// TIA Portal V20 export
// export: Created 2025-12-01T14:56:58.9383901Z, ExportSetting None, DisplayName Totally Integrated Automation Portal, DisplayVersion V20 Update 3, DisplayName TIA Portal Openness, DisplayVersion V20 Update 3, DisplayName TIA Portal Version Control Interface, DisplayVersion V20 Update 3, DisplayName STEP 7 Professional, DisplayVersion V20 Update 3, DisplayName STEP 7 Safety, DisplayVersion V20 Update 2, DisplayName WinCC Basic/Comfort/Advanced, DisplayVersion V20 Update 3, DisplayName WinCC Professional, DisplayVersion V20 Update 3, DisplayName WinCC Unified, DisplayVersion V20 Update 3
FUNCTION_BLOCK "FB89_GALIBO_Remontada_EnRodillos"   // FB89, LAD
TITLE = Galibo de 5 Alturas (2023)
{ S7_Optimized_Access := 'FALSE' }
AUTHOR : GALIBO
NAME : 20140101
VERSION : 3.0
// stored: AutoNumber false, SetENOAutomatically false
   VAR_INPUT
      Mesa : UInt;
      NumGalibo : UInt;
      pHs_Remontado_1Dcha : Bool;
      pHs_Remontado_2Dcha : Bool;
      pHs_Remontado_1Izq : Bool;
      pHs_Remontado_2Izq : Bool;
      HabilitarLectura : Bool;
      PermisoLectura : Bool;
      Rearmar_ConMesaLibre : Bool;
      V_Estabilidad : Int;
   END_VAR
   VAR_OUTPUT
      Codigo : Word;
      FinLectura : Bool;
   END_VAR
   VAR_IN_OUT
      SinopticoGalibo_Señal : "UDT_HMI_SeñalesGalibo";
      SinopticoGalibo_Codigo : Word;
   END_VAR
   VAR
      CNT_Estabilidad : "FB910_CNT_UHS";
      GAL_ET00 : Bool;
      GAL_ET01 : Bool;
      GAL_ET02 : Bool;
      GAL_ET03 : Bool;
      pHsGalibo_OK { ExternalAccessible := 'False'; ExternalVisible := 'False'; ExternalWritable := 'False'} : Bool;
      LeerRemontado : Bool;
      FinRemontado : Bool;
      Remontado_NO : Bool;
      Remontado_SI : Bool;
      CodigoRemontado : SInt;
      MemoCodigo : Word;
      STAT_Baliza_Galibo : Bool;
   END_VAR
   VAR_TEMP
      EstadoZona : "EstadoZona";
      EstadoVI : "EstadosMesa";
   END_VAR
BEGIN

REGION Network 1: INICIALIZAR - Recoger las Variables de Estado de la Mesa
   // Se recoge - Estado_CBx
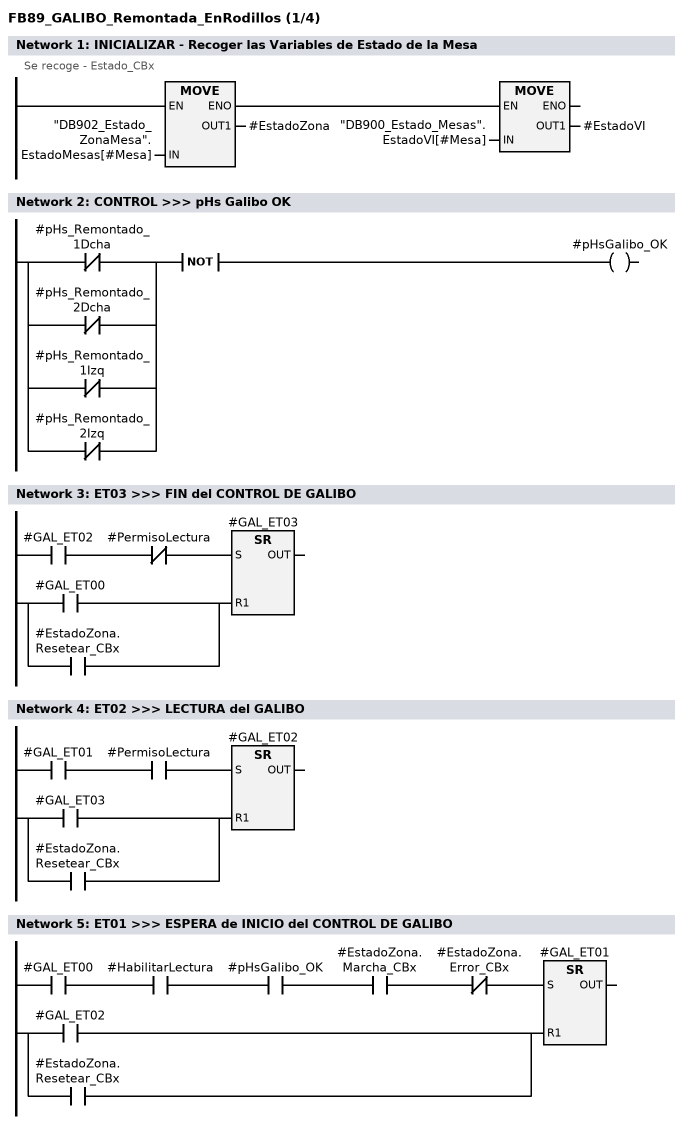
   RUNG wire#powerrail
      Move(in := "DB902_Estado_ZonaMesa".EstadoMesas[#Mesa], out1 => #EstadoZona)
      Move(in := "DB900_Estado_Mesas".EstadoVI[#Mesa], out1 => #EstadoVI)
   END_RUNG
   // the same network as SCL:
   #EstadoZona := "DB902_Estado_ZonaMesa".EstadoMesas[#Mesa];
   #EstadoVI := "DB900_Estado_Mesas".EstadoVI[#Mesa];
END_REGION

REGION Network 2: CONTROL >>> pHs Galibo OK
   RUNG wire#powerrail
      I_Contact( #pHs_Remontado_1Dcha )
      wire#w1
      Not()
      Coil( #pHsGalibo_OK )
   END_RUNG
   RUNG wire#powerrail
      I_Contact( #pHs_Remontado_2Dcha )
   END_RUNG wire#w1
   RUNG wire#powerrail
      I_Contact( #pHs_Remontado_1Izq )
   END_RUNG wire#w1
   RUNG wire#powerrail
      I_Contact( #pHs_Remontado_2Izq )
   END_RUNG wire#w1
   // the same network as SCL:
   #pHsGalibo_OK := NOT (NOT #pHs_Remontado_1Dcha OR NOT #pHs_Remontado_2Dcha OR NOT #pHs_Remontado_1Izq OR NOT #pHs_Remontado_2Izq);
END_REGION

REGION Network 3: ET03 >>> FIN del CONTROL DE GALIBO
   RUNG wire#powerrail
      Contact( #GAL_ET02 )
      I_Contact( #PermisoLectura )
      S_SR(operand := #GAL_ET03, r1 := wire#w1)
   END_RUNG
   RUNG wire#powerrail
      Contact( #GAL_ET00 )
   END_RUNG wire#w1
   RUNG wire#powerrail
      Contact( #EstadoZona.Resetear_CBx )
   END_RUNG wire#w1
   // the same network as SCL:
   IF #GAL_ET02 AND NOT #PermisoLectura THEN
       #GAL_ET03 := TRUE;   // SR flip-flop
   END_IF;
   IF #GAL_ET00 OR #EstadoZona.Resetear_CBx THEN #GAL_ET03 := FALSE; END_IF;
END_REGION

REGION Network 4: ET02 >>> LECTURA del GALIBO
   RUNG wire#powerrail
      Contact( #GAL_ET01 )
      Contact( #PermisoLectura )
      S_SR(operand := #GAL_ET02, r1 := wire#w1)
   END_RUNG
   RUNG wire#powerrail
      Contact( #GAL_ET03 )
   END_RUNG wire#w1
   RUNG wire#powerrail
      Contact( #EstadoZona.Resetear_CBx )
   END_RUNG wire#w1
   // the same network as SCL:
   IF #GAL_ET01 AND #PermisoLectura THEN
       #GAL_ET02 := TRUE;   // SR flip-flop
   END_IF;
   IF #GAL_ET03 OR #EstadoZona.Resetear_CBx THEN #GAL_ET02 := FALSE; END_IF;
END_REGION

REGION Network 5: ET01 >>> ESPERA de INICIO del CONTROL DE GALIBO
   RUNG wire#powerrail
      Contact( #GAL_ET00 )
      Contact( #HabilitarLectura )
      Contact( #pHsGalibo_OK )
      Contact( #EstadoZona.Marcha_CBx )
      I_Contact( #EstadoZona.Error_CBx )
      S_SR(operand := #GAL_ET01, r1 := wire#w1)
   END_RUNG
   RUNG wire#powerrail
      Contact( #GAL_ET02 )
   END_RUNG wire#w1
   RUNG wire#powerrail
      Contact( #EstadoZona.Resetear_CBx )
   END_RUNG wire#w1
   // the same network as SCL:
   IF #GAL_ET00 AND #HabilitarLectura AND #pHsGalibo_OK AND #EstadoZona.Marcha_CBx AND NOT #EstadoZona.Error_CBx THEN
       #GAL_ET01 := TRUE;   // SR flip-flop
   END_IF;
   IF #GAL_ET02 OR #EstadoZona.Resetear_CBx THEN #GAL_ET01 := FALSE; END_IF;
END_REGION

REGION Network 6: ET00 >>> INICIO
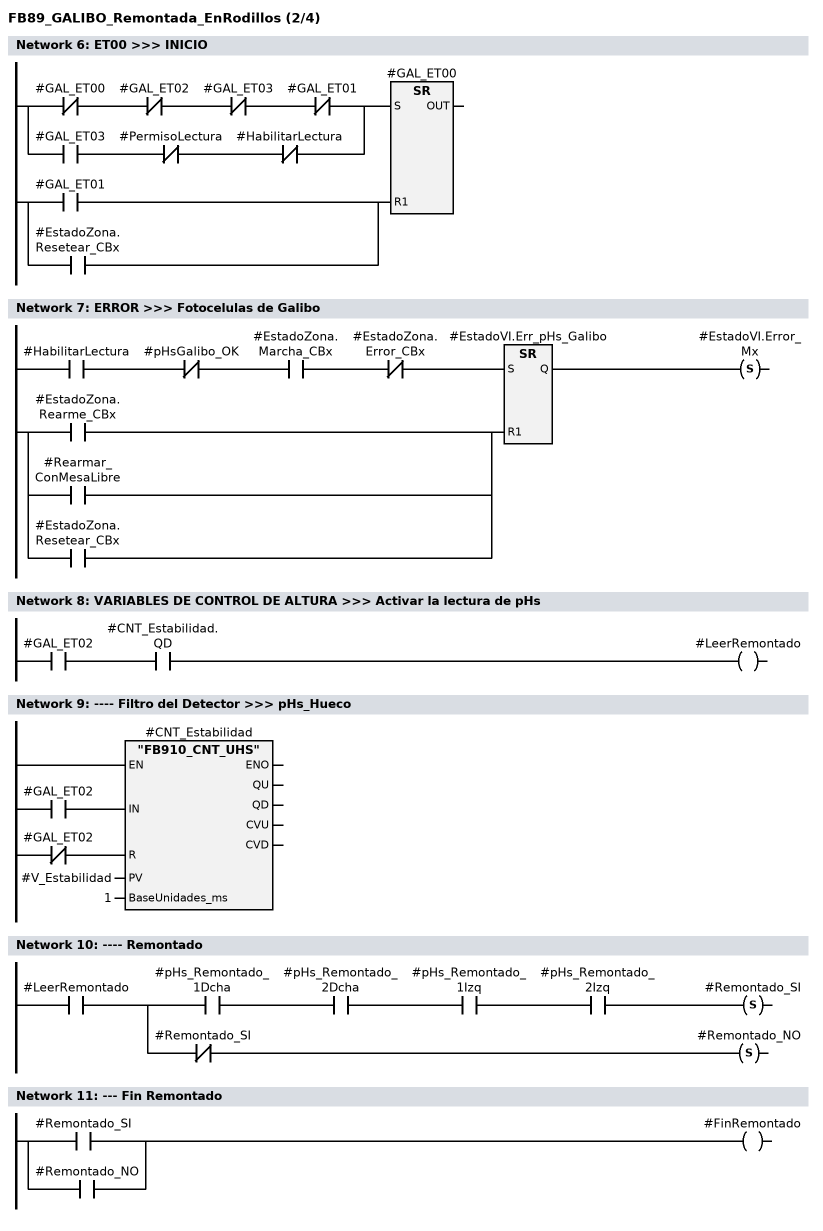
   RUNG wire#powerrail
      I_Contact( #GAL_ET00 )
      I_Contact( #GAL_ET02 )
      I_Contact( #GAL_ET03 )
      I_Contact( #GAL_ET01 )
      wire#w1
      S_SR(operand := #GAL_ET00, r1 := wire#w2)
   END_RUNG
   RUNG wire#powerrail
      Contact( #GAL_ET03 )
      I_Contact( #PermisoLectura )
      I_Contact( #HabilitarLectura )
   END_RUNG wire#w1
   RUNG wire#powerrail
      Contact( #GAL_ET01 )
   END_RUNG wire#w2
   RUNG wire#powerrail
      Contact( #EstadoZona.Resetear_CBx )
   END_RUNG wire#w2
   // the same network as SCL:
   IF (NOT #GAL_ET00 AND NOT #GAL_ET02 AND NOT #GAL_ET03 AND NOT #GAL_ET01) OR (#GAL_ET03 AND NOT #PermisoLectura AND NOT #HabilitarLectura) THEN
       #GAL_ET00 := TRUE;   // SR flip-flop
   END_IF;
   IF #GAL_ET01 OR #EstadoZona.Resetear_CBx THEN #GAL_ET00 := FALSE; END_IF;
END_REGION

REGION Network 7: ERROR >>> Fotocelulas de Galibo
   RUNG wire#powerrail
      Contact( #HabilitarLectura )
      I_Contact( #pHsGalibo_OK )
      Contact( #EstadoZona.Marcha_CBx )
      I_Contact( #EstadoZona.Error_CBx )
      S_SR(operand := #EstadoVI.Err_pHs_Galibo, r1 := wire#w1)
      S_Coil( #EstadoVI.Error_Mx )
   END_RUNG
   RUNG wire#powerrail
      Contact( #EstadoZona.Rearme_CBx )
   END_RUNG wire#w1
   RUNG wire#powerrail
      Contact( #Rearmar_ConMesaLibre )
   END_RUNG wire#w1
   RUNG wire#powerrail
      Contact( #EstadoZona.Resetear_CBx )
   END_RUNG wire#w1
   // the same network as SCL:
   IF #HabilitarLectura AND NOT #pHsGalibo_OK AND #EstadoZona.Marcha_CBx AND NOT #EstadoZona.Error_CBx THEN
       #EstadoVI.Err_pHs_Galibo := TRUE;   // SR flip-flop
   END_IF;
   IF #EstadoZona.Rearme_CBx OR #Rearmar_ConMesaLibre OR #EstadoZona.Resetear_CBx THEN
       #EstadoVI.Err_pHs_Galibo := FALSE;
   END_IF;
   IF #EstadoVI.Err_pHs_Galibo THEN #EstadoVI.Error_Mx := TRUE; END_IF;
END_REGION

REGION Network 8: VARIABLES DE CONTROL DE ALTURA >>> Activar la lectura de pHs
   RUNG wire#powerrail
      Contact( #GAL_ET02 )
      Contact( #CNT_Estabilidad.QD )
      Coil( #LeerRemontado )
   END_RUNG
   // the same network as SCL:
   #LeerRemontado := #GAL_ET02 AND #CNT_Estabilidad.QD;
END_REGION

REGION Network 9: ---- Filtro del Detector >>> pHs_Hueco
   RUNG wire#powerrail
      #CNT_Estabilidad(IN := wire#w1, R := wire#w2, PV := #V_Estabilidad, BaseUnidades_ms := 1, QU =>, QD =>, CVU =>, CVD =>)
   END_RUNG
   RUNG wire#powerrail
      Contact( #GAL_ET02 )
   END_RUNG wire#w1
   RUNG wire#powerrail
      I_Contact( #GAL_ET02 )
   END_RUNG wire#w2
   // the same network as SCL:
   #CNT_Estabilidad(IN := #GAL_ET02, R := NOT #GAL_ET02, PV := #V_Estabilidad, BaseUnidades_ms := 1);   // "FB910_CNT_UHS"
END_REGION

REGION Network 10: ---- Remontado
   RUNG wire#powerrail
      Contact( #LeerRemontado )
      wire#w1
      Contact( #pHs_Remontado_1Dcha )
      Contact( #pHs_Remontado_2Dcha )
      Contact( #pHs_Remontado_1Izq )
      Contact( #pHs_Remontado_2Izq )
      S_Coil( #Remontado_SI )
   END_RUNG
   RUNG wire#w1
      I_Contact( #Remontado_SI )
      S_Coil( #Remontado_NO )
   END_RUNG
   // the same network as SCL:
   IF #LeerRemontado AND #pHs_Remontado_1Dcha AND #pHs_Remontado_2Dcha AND #pHs_Remontado_1Izq AND #pHs_Remontado_2Izq THEN
       #Remontado_SI := TRUE;
   END_IF;
   IF #LeerRemontado AND NOT #Remontado_SI THEN #Remontado_NO := TRUE; END_IF;
END_REGION

REGION Network 11: --- Fin Remontado
   RUNG wire#powerrail
      Contact( #Remontado_SI )
      wire#w1
      Coil( #FinRemontado )
   END_RUNG
   RUNG wire#powerrail
      Contact( #Remontado_NO )
   END_RUNG wire#w1
   // the same network as SCL:
   #FinRemontado := #Remontado_SI OR #Remontado_NO;
END_REGION

REGION Network 12: --- Rearme
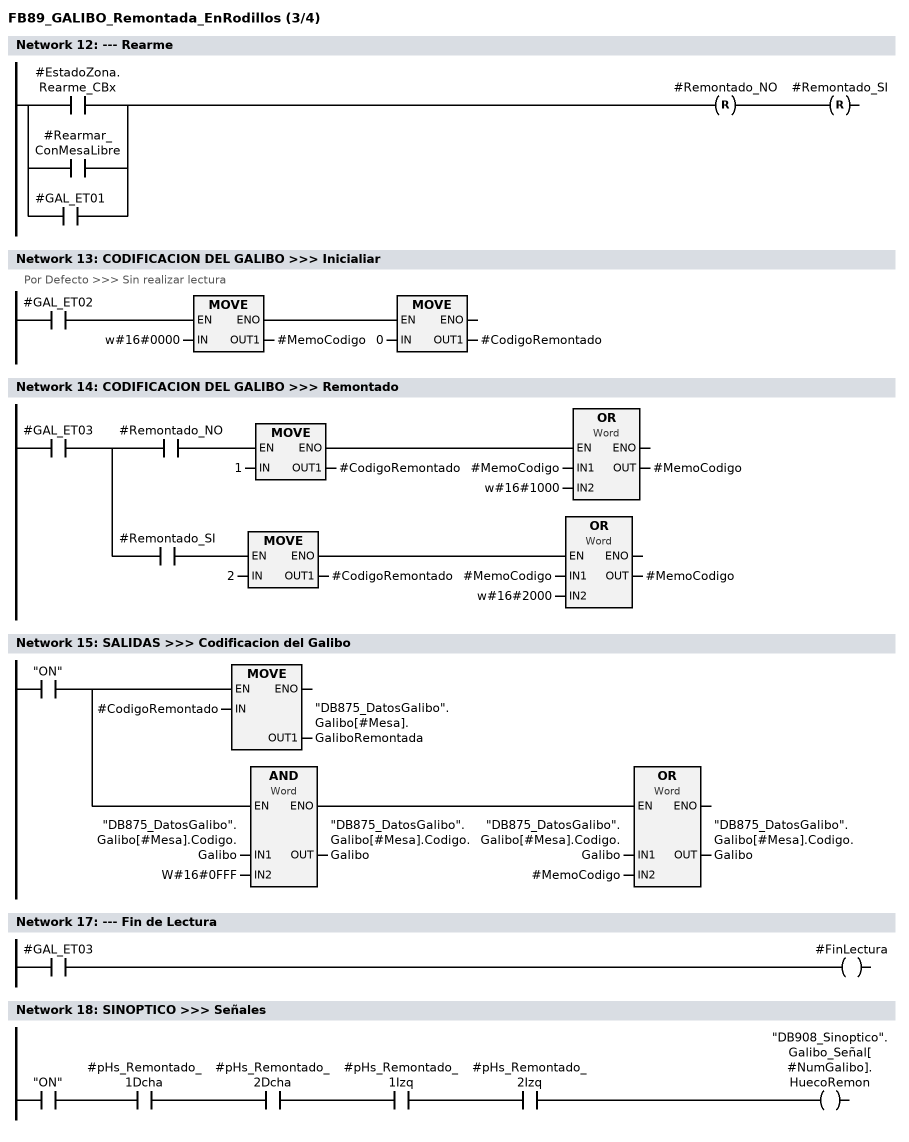
   RUNG wire#powerrail
      Contact( #EstadoZona.Rearme_CBx )
      wire#w1
      R_Coil( #Remontado_NO )
      R_Coil( #Remontado_SI )
   END_RUNG
   RUNG wire#powerrail
      Contact( #Rearmar_ConMesaLibre )
   END_RUNG wire#w1
   RUNG wire#powerrail
      Contact( #GAL_ET01 )
   END_RUNG wire#w1
   // the same network as SCL:
   IF #EstadoZona.Rearme_CBx OR #Rearmar_ConMesaLibre OR #GAL_ET01 THEN
       #Remontado_NO := FALSE;
       #Remontado_SI := FALSE;
   END_IF;
END_REGION

REGION Network 13: CODIFICACION DEL GALIBO >>> Inicialiar
   // Por Defecto >>> Sin realizar lectura
   RUNG wire#powerrail
      Contact( #GAL_ET02 )
      { S7_GenerateENO := "TRUE" } Move(in := w#16#0000, out1 => #MemoCodigo)
      { S7_GenerateENO := "TRUE" } Move(in := 0, out1 => #CodigoRemontado)
   END_RUNG
   // the same network as SCL:
   // ENO of a box is taken as its EN; it also drops when the box reports an error
   IF #GAL_ET02 THEN
       #MemoCodigo := w#16#0000;
       #CodigoRemontado := 0;
   END_IF;
END_REGION

REGION Network 14: CODIFICACION DEL GALIBO >>> Remontado
   // ENO of a box is taken as its EN; it also drops when the box reports an error
   IF #GAL_ET03 AND #Remontado_NO THEN
       #CodigoRemontado := 1;
       #MemoCodigo := #MemoCodigo OR w#16#1000;
   END_IF;
   IF #GAL_ET03 AND #Remontado_SI THEN
       #CodigoRemontado := 2;
       #MemoCodigo := #MemoCodigo OR w#16#2000;
   END_IF;
END_REGION

REGION Network 15: SALIDAS >>> Codificacion del Galibo
   IF "ON" THEN
       "DB875_DatosGalibo".Galibo[#Mesa].GaliboRemontada := #CodigoRemontado;
       "DB875_DatosGalibo".Galibo[#Mesa].Codigo.Galibo := "DB875_DatosGalibo".Galibo[#Mesa].Codigo.Galibo AND W#16#0FFF;
       "DB875_DatosGalibo".Galibo[#Mesa].Codigo.Galibo := "DB875_DatosGalibo".Galibo[#Mesa].Codigo.Galibo OR #MemoCodigo;
   END_IF;
END_REGION

REGION Network 16: ---- Aviso de Error NOTA >>> NO PROCEDE
END_REGION

REGION Network 17: --- Fin de Lectura
   RUNG wire#powerrail
      Contact( #GAL_ET03 )
      Coil( #FinLectura )
   END_RUNG
   // the same network as SCL:
   #FinLectura := #GAL_ET03;
END_REGION

REGION Network 18: SINOPTICO >>> Señales
   RUNG wire#powerrail
      Contact( "ON" )
      Contact( #pHs_Remontado_1Dcha )
      Contact( #pHs_Remontado_2Dcha )
      Contact( #pHs_Remontado_1Izq )
      Contact( #pHs_Remontado_2Izq )
      Coil( "DB908_Sinoptico".Galibo_Señal[#NumGalibo].HuecoRemon )
   END_RUNG
   // the same network as SCL:
   "DB908_Sinoptico".Galibo_Señal[#NumGalibo].HuecoRemon := "ON" AND #pHs_Remontado_1Dcha AND #pHs_Remontado_2Dcha AND #pHs_Remontado_1Izq AND #pHs_Remontado_2Izq;
END_REGION

REGION Network 19: SINOPTICO >>> Codigo
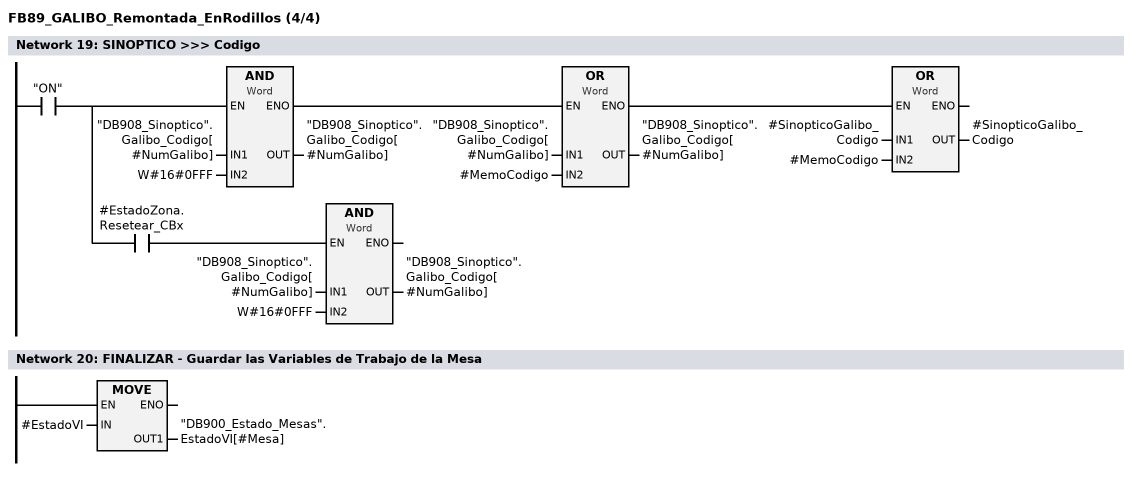
   IF "ON" THEN
       "DB908_Sinoptico".Galibo_Codigo[#NumGalibo] := "DB908_Sinoptico".Galibo_Codigo[#NumGalibo] AND W#16#0FFF;
       "DB908_Sinoptico".Galibo_Codigo[#NumGalibo] := "DB908_Sinoptico".Galibo_Codigo[#NumGalibo] OR #MemoCodigo;
       #SinopticoGalibo_Codigo := #SinopticoGalibo_Codigo OR #MemoCodigo;
   END_IF;
   IF "ON" AND #EstadoZona.Resetear_CBx THEN
       "DB908_Sinoptico".Galibo_Codigo[#NumGalibo] := "DB908_Sinoptico".Galibo_Codigo[#NumGalibo] AND W#16#0FFF;
   END_IF;
END_REGION

REGION Network 20: FINALIZAR - Guardar las Variables de Trabajo de la Mesa
   RUNG wire#powerrail
      Move(in := #EstadoVI, out1 => "DB900_Estado_Mesas".EstadoVI[#Mesa])
   END_RUNG
   // the same network as SCL:
   "DB900_Estado_Mesas".EstadoVI[#Mesa] := #EstadoVI;
END_REGION
END_FUNCTION_BLOCK
